// TIA Portal V18 export
TYPE "PLCtoMES_RealTimeData"
// stored: IsFailsafeCompliant false
   STRUCT
      "P-RealTimeData" { S7_SetPoint := 'True'} : Array[1..64] of "PLCtoMES_ProcessData";
      Reserve { S7_SetPoint := 'True'} : Array[1..100] of Byte;
   END_STRUCT;
END_TYPE
